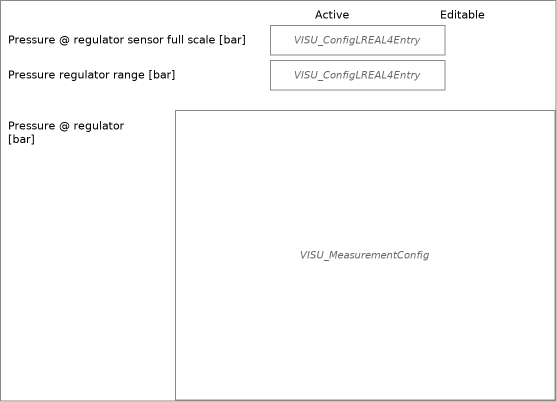
VISUALIZATION VISU_M1Config_Radial_RegulatorPressure  // 557x402
VAR_IN_OUT
    editable : M1RadialSupportConfig;
	active : M1RadialSupportConfig;
END_VAR
    Label (270,5 125x20), "Active"
    Label (400,5 125x20), "Editable"
    Label (5,25 260x30), "Pressure @ regulator sensor full scale [bar]"
    Frame (270,25 175x30)
        shows VISU_ConfigLREAL4Entry(active := active.regulatorPressureSensorFullScale, editable := editable.regulatorPressureSensorFullScale)
    Label (5,100 145x65), "Pressure @ regulator [bar]"
    Label (5,60 260x30), "Pressure regulator range [bar]"
    Frame (270,60 175x30)
        shows VISU_ConfigLREAL4Entry(active := active.pressureRegulatorRange, editable := editable.pressureRegulatorRange)
    Frame (175,110 380x290)
        shows VISU_MeasurementConfig(active := active.regulatorPressure, editable := editable.regulatorPressure)
END_VISUALIZATION

(* stored: Version 1.1.0.1, ProductVersion 3.1.4019.2
   Visu VISU_M1Config_Radial_RegulatorPressure: Id {e6022e26-af9f-429b-918c-242672c34eab} *)
